// TIA Portal V17 export
// export: Created 2022-04-06T07:28:39.1030181Z, ExportSetting WithDefaults, DisplayName Totally Integrated Automation Portal, DisplayVersion V17, DisplayName TIA Portal Openness, DisplayVersion V17, DisplayName TIA Portal Version Control Interface, DisplayVersion V17, DisplayName TIA Portal Test Suite Advanced, DisplayVersion V17, DisplayName SINAMICS Startdrive Advanced, DisplayVersion V17, DisplayName SINAMICS Startdrive G130, G150, S120, S150, SINAMICS MV, S210, DisplayVersion V17, DisplayName SINAMICS Startdrive G110M, G120, G120C, G120D, G120P, G115D, DisplayVersion V17, DisplayName STEP 7 Professional, DisplayVersion V17, DisplayName STEP 7 Safety, DisplayVersion V17, DisplayName WinCC Advanced / Unified PC, DisplayVersion V17
DATA_BLOCK "InstDataLogNewFile"   // DB13
VERSION : 0.1
// stored: AutoNumber true, DBAccessibleFromOPCUA true, DBAccessibleFromWebserver true, InstanceOfName DataLog1500, InstanceOfType FB
"DataLog1500"
   // VAR_INPUT
   //    write : Bool;
   //    records : UDInt;
   //    timestamp : UInt;
   //    "name" : String;
   //    header : String;
   //    clear : Bool;
   //    newFileMax : USInt;
   //    delete : Bool;
   // END_VAR
   // VAR_OUTPUT
   //    done { ExternalWritable := 'False'} : Bool;
   //    busy { ExternalWritable := 'False'} : Bool;
   //    error { ExternalWritable := 'False'} : Bool;
   //    status { ExternalWritable := 'False'} : Word;
   //    subFunctionStatus { ExternalWritable := 'False'} : Word;
   //    id { ExternalWritable := 'False'} : DWord;
   //    numberRecords { ExternalWritable := 'False'} : UDInt;
   //    sync { ExternalWritable := 'False'} : Bool;
   //    full { ExternalWritable := 'False'} : Bool;
   //    currentName { ExternalWritable := 'False'} : String;
   // END_VAR
   // VAR_IN_OUT
   //    data : Variant;
   // END_VAR
   // VAR RETAIN
   //    statId { ExternalAccessible := 'False'; ExternalVisible := 'False'; ExternalWritable := 'False'} : DWord;
   //    statNumberRecords { ExternalAccessible := 'False'; ExternalVisible := 'False'; ExternalWritable := 'False'} : UDInt;
   //    statSync { ExternalAccessible := 'False'; ExternalVisible := 'False'; ExternalWritable := 'False'} : Bool;
   //    statFull { ExternalAccessible := 'False'; ExternalVisible := 'False'; ExternalWritable := 'False'} : Bool;
   //    statClosed { ExternalAccessible := 'False'; ExternalVisible := 'False'; ExternalWritable := 'False'} : Bool;
   //    statFileNumber { ExternalAccessible := 'False'; ExternalVisible := 'False'; ExternalWritable := 'False'} : USInt;
   //    statName { ExternalAccessible := 'False'; ExternalVisible := 'False'; ExternalWritable := 'False'} : String;
   // END_VAR
   // VAR
   //    statDelete { ExternalAccessible := 'False'; ExternalVisible := 'False'; ExternalWritable := 'False'} : Bool;
   //    statWriteOld { ExternalAccessible := 'False'; ExternalVisible := 'False'; ExternalWritable := 'False'} : Bool;
   //    statDeleteOld { ExternalAccessible := 'False'; ExternalVisible := 'False'; ExternalWritable := 'False'} : Bool;
   //    statDone { ExternalAccessible := 'False'; ExternalVisible := 'False'; ExternalWritable := 'False'} : Bool;
   //    statBusy { ExternalAccessible := 'False'; ExternalVisible := 'False'; ExternalWritable := 'False'} : Bool;
   //    statError { ExternalAccessible := 'False'; ExternalVisible := 'False'; ExternalWritable := 'False'} : Bool;
   //    statStatus { ExternalAccessible := 'False'; ExternalVisible := 'False'; ExternalWritable := 'False'} : Word;
   //    statSubfunctionStatus { ExternalAccessible := 'False'; ExternalVisible := 'False'; ExternalWritable := 'False'} : Word;
   //    statFBState { ExternalAccessible := 'False'; ExternalVisible := 'False'; ExternalWritable := 'False'} : DInt;
   //    instDataLogCreate { ExternalAccessible := 'False'; ExternalVisible := 'False'; ExternalWritable := 'False'} : DataLogCreate;
   //    instDataLogOpen { ExternalAccessible := 'False'; ExternalVisible := 'False'; ExternalWritable := 'False'} : DataLogOpen;
   //    instDataLogWrite { ExternalAccessible := 'False'; ExternalVisible := 'False'; ExternalWritable := 'False'} : DataLogWrite;
   //    instDataLogClear { ExternalAccessible := 'False'; ExternalVisible := 'False'; ExternalWritable := 'False'} : DataLogClear;
   //    instDataLogClose { ExternalAccessible := 'False'; ExternalVisible := 'False'; ExternalWritable := 'False'} : DataLogClose;
   //    instDataLogNewFile { ExternalAccessible := 'False'; ExternalVisible := 'False'; ExternalWritable := 'False'} : DataLogNewFile;
   //    instDataLogDelete { ExternalAccessible := 'False'; ExternalVisible := 'False'; ExternalWritable := 'False'} : DataLogDelete;
   // END_VAR
BEGIN
END_DATA_BLOCK
